(* IEC 61131-3 sources: volt/packages/volt-lsp-iec/test-corpus/bakon-nano/Device/Plc Logic/Application/Global Variables, 9 files *)

(* ---- CAN_TO_PLC.gvl ---- *)
//This gobal variable list is received via the network.
//Sender: Imported from file '\\SRV2012\Home$\pieter\Documents\Projecten\P10037 Hert nano met wasbak\21000149 Software\CAN Bridge\CAN_TO_PLC.gvl'
//Protocol: UDP

{attribute 'qualified_only'}
VAR_GLOBAL
	dwAGM1_PowerLoss			: DWORD;
	rAGM1_Frequency				: REAL;
	bAGM1_CommFailure			: BOOL;
	dwErrorDetailsAGM1			: DWORD;
	bUltrasonic1				: BOOL;
END_VAR
%CLASS NVL
%NETVAR ImportFromFile: true
%NETVAR ImportFileName: \\SRV2012\Home$\pieter\Documents\Projecten\P10037 Hert nano met wasbak\21000149 Software\CAN Bridge\CAN_TO_PLC.gvl
%NETVAR TaskName: LogicTask
%NETVAR SenderGVLName: ''
%NETVAR ImportNetVarProperties.Acknowledge: false
%NETVAR ImportNetVarProperties.Checksum: false
%NETVAR ImportNetVarProperties.EventVariable: ''
%NETVAR ImportNetVarProperties.Interval: T#50ms
%NETVAR ImportNetVarProperties.ListIdentifier: 2
%NETVAR ImportNetVarProperties.MinimumGap: T#20ms
%NETVAR ImportNetVarProperties.PackVariables: true
%NETVAR ImportNetVarProperties.ProtocolName: UDP
%NETVAR ImportNetVarProperties.TransmitCyclic: true
%NETVAR ImportNetVarProperties.TransmitOnChange: false
%NETVAR ImportNetVarProperties.TransmitOnEvent: false
%NETVAR ImportNetVarProperties.TaskName: LogicTask
%NETVAR ImportNetVarProperties.ImportFileName: ''
%NETVAR ImportNetVarProperties.ProtocolParameterValues: UDP=Broadcast Adr.=192.168.27.230; Port=1202

(* ---- Global_Constantes_MachineDependant.gvl ---- *)
VAR_GLOBAL CONSTANT

(*********************** AFHANKELIJK VAN MACHINE!! ***********************)

	C_LimitKnifeStrokeMax		: REAL := 225;		(* Controle of machine parameter tussen de limieten valt *)
	C_LimitKnifeStrokeMin		: REAL := 60;		(* (controle of mach par goed opgeslagen zijn) *)

	C_rTargetX_TableCheck		: REAL := 2.1;		(* x positie voor de tafel sensor controle *)
	C_rXAxis_SafeCleaningPos	: REAL := 3;		(* x positie voor de tafel veilig om waterbakje omhoog te sturen *)

	C_rExtraMarginKnifeHeight	: REAL := 8;		(* extra starthoogte van het mes bovenop de gewenste producthoogte *)

	C_rMinOvershootX			: REAL	:= 3;		(* minimaal 1 meer dan de negatieve sw limit *)
	C_rMaxOvershootX			: REAL	:= 683;//688	(* minimaal 1 minder dan de positieve sw limit *)
	C_rMaxOvershootX_XL			: REAL  := 898;		(* voor XL Machine*)
	C_rMinOvershootY			: REAL	:= 3;		(* minimaal 1 meer dan de negatieve sw limit *)
	C_rMaxOvershootY			: REAL	:= 488;		(* minimaal 1 minder dan de positieve sw limit *)
	C_rMaxOvershootY_XL			: REAL  := 658;

	C_rMinimumTrimSlab		: REAL	:= 0;
	C_rMaxPowerUS1			: REAL	:= 100;		(* value from 50 to 100 % *)

	(********************************************* Other  Constantes *********************************************)
	C_rPi								: REAL	:= 3.14159265358979;

	C_wNumberOfMotionObjects	: INT := 1600;

	C_NOT_ACTIVE  				:INT	:=  -1;
	C_INITIAL      					:INT	:=   0;
	C_WAIT_EXEC  	  			:INT	:=	995;
	C_INITIALISE   				:INT 	:=	996;
	C_STOPPED      				:INT	:=	997;
	C_READY        				:INT	:=	998;
	C_LAST       	  				:INT	:=	999;

END_VAR

(* ---- Global_Variables.gvl ---- *)
	VAR_GLOBAL
	g_sMACH							: sMACH_DATA;

	g_bCMD_US_Start1				: BOOL;
	g_bCMD_US_Test1					: BOOL;
	g_bUS_EnableRV					: BOOL;		(* Enable US generator when knife is in product *)
	g_bUS_EnableCleaning			: BOOL;		(* Enable US generator during cleaning *)

	g_bSaveMachPar					: BOOL;		(* Save Mach par aan einde van automaat *)

	ModusRV							: sModusRondVierkant;

	g_uParRondVierkant				: strRondVierkantParameters;

	g_bFirstCycle					: BOOL;
	g_bOnDelayed					: BOOL;

	g_bCalculationStart				: BOOL;
	g_bCalculationDone				: BOOL;
	g_bSUB_CleanKnifeStart			: BOOL;
	g_bSUB_CleanKnifeDone			: BOOL;
	g_bCleanRequest					: BOOL;

	g_bSUB_InitStart				: BOOL;
	g_bSUB_InitDone					: BOOL;

	g_bProductNotFinished			: BOOL;	(* cuts on product not completed *)

	g_bHomingDone					: BOOL;

	g_bTestAGM1						: BOOL;
	g_bResetMaster					: BOOL;
	(* Machine configuration bits *)
	gMachConfig						: sMach_Setup;
	gProductOption					: sProd_Setup;

	(* Ultrasonic variables *)
	//g_dwAGM1_Status					: DWORD;
	g_dwAGM1_PowerLoss				: DWORD;
	g_rAGM1_Frequency				: REAL;

	g_sCalculated					: sMACH_Calculated;
	g_aCuttingPositions				: ARRAY [1..C_wNumberOfMotionObjects] OF XYA_Target;
	g_sCuttingPositionsInfo			: ArrayInfo;
	g_aWastePositions				: ARRAY [1..100] OF XYA_Target;
	g_sWastePositionsInfo			: ArrayInfo;

	g_bTrimFront					: BOOL;	(* Variable used in calculation functions*)
	g_bTrimRear						: BOOL;	(* Variable used in calculation functions*)
	g_bTrimLeft						: BOOL;	(* Variable used in calculation functions*)
	g_bTrimRight					: BOOL;	(* Variable used in calculation functions*)
	g_rDistanceBetweenCuts_InX		: REAL;	(* Variable used in calculation functions*)
	g_rDistanceBetweenCuts_InY		: REAL;	(* Variable used in calculation functions*)
	g_rHoekInRad					: REAL;	(* Variable used in calculation functions*)
	g_rHoekInRad2					: REAL;	(* Variable used in calculation functions*)
	g_rEndTargetX					: REAL;	(* Variable used for saving end target*)
	g_rEndTargetY					: REAL;	(* Variable used for saving end target*)
	g_rEndTargetA					: REAL;	(* Variable used for saving end target*)
	g_rEndTargetK					: REAL;	(* Variable used for saving end target*)

	g_bCurrentTableUniversal10		: BOOL := FALSE;

	g_sMCHCopyMade					: BOOL := FALSE;
	g_sMCHParCopy					: sMACH_MACH_Parameters;
	g_sRCPCopyMade					: BOOL := FALSE;
	g_sRCPParCopy					: sMACH_RCP_Parameters;
	{warning 'Disabled for compatibility - SVE'}
	//g_Logger						: PLC_Logger;
END_VAR

(* ---- PLC_TO_CAN.gvl ---- *)
{attribute 'qualified_only'}
VAR_GLOBAL
	g_bOnDelayed 			: BOOL;
	g_bDQ_Ultrasonic1 		: BOOL;
	g_bTestAGM1 			: BOOL;
	g_HMI_MCH_Parameters	: sMACH_MACH_Parameters;
	g_HMI_RCP_Parameters	: sMACH_RCP_Parameters;
	g_HMI_MachCommand		: sMACH_HMI_UnitCmd;
	C_rMaxPowerUS1			: REAL;
END_VAR
%NETVAR Acknowledge: false
%NETVAR Checksum: false
%NETVAR EventVariable: ''
%NETVAR Interval: T#50ms
%NETVAR ListIdentifier: 1
%NETVAR MinimumGap: T#20ms
%NETVAR PackVariables: true
%NETVAR ProtocolName: UDP
%NETVAR TransmitCyclic: true
%NETVAR TransmitOnChange: false
%NETVAR TransmitOnEvent: false
%NETVAR TaskName: LogicTask
%NETVAR ImportFileName: ''
%NETVAR ProtocolParameterValues: UDP=Broadcast Adr.=192.168.27.231; Port=1202
%FILE_LINK ExportBeforeCompile '\\SRV2012\Home$$\pieter\Documents\Projecten\P10037 Hert nano met wasbak\21000149 Software\PLC\PLC_TO_CAN.gvl'

(* ---- VAR_AxisControl_ECSEP.gvl ---- *)
VAR_GLOBAL
	g_uControl_X_Axis		:KC_AxisBasicsControl;	(* VIRTUAL AXIS *)
	g_uStatus_X_Axis			:KC_AxisBasicsStatus;	(* VIRTUAL AXIS *)
	g_uControl_Y_Axis		:KC_AxisBasicsControl;	(* VIRTUAL AXIS *)
	g_uStatus_Y_Axis			:KC_AxisBasicsStatus;	(* VIRTUAL AXIS *)
	g_uControl_Front_Axis	:KC_AxisBasicsControl;
	g_uStatus_Front_Axis	:KC_AxisBasicsStatus;
	g_uControl_Rear_Axis	:KC_AxisBasicsControl;
	g_uStatus_Rear_Axis		:KC_AxisBasicsStatus;
	g_uControl_Z_Axis		:KC_AxisBasicsControl;
	g_uStatus_Z_Axis			:KC_AxisBasicsStatus;
	g_uControl_R_Axis		:KC_AxisBasicsControl;
	g_uStatus_R_Axis		:KC_AxisBasicsStatus;
END_VAR

(* ---- VAR_HMI.gvl ---- *)
VAR_GLOBAL
	(* Communicatie met VisiwinNet Visualisatie Professional V6.3 *)
	g_HMI_MachCommand					: sMACH_HMI_UnitCmd;

	g_HMI_bRecipeIsReset		: BOOL;

	(*status variables *)
	g_sHMI_Mach_UnitStatus				:sMACH_HMI_UnitStatus;				(*module status variables*)

	(* Counters *)
	g_sHMI_CountersDay					: sCounters;		(* all day counters *)

	g_sHMI_ScanData					: sScanData;	(*Data for max follow/torque scan of machine*)

	(* Data for new visu *)
	g_sHMI_VisuCutsArray	: ARRAY[1..150] OF VisuCut;
	g_sHMI_NewRecipeName			: STRING;
	g_bHMI_UseExistingRecipe		:BOOL;
	g_sHMI_FromCecipeName			: STRING;
	g_sHMI_MachParName				: STRING;
	g_sHMI_RcpClmns					: ClmnChoices;
	g_sHMI_Recipe_Clmn1_Choice	: INT; // SlabRound = 1, SlabRound with fingers = 2, Tray = 3
	g_sHMI_Recipe_Clmn2_Choice	: INT; //
	g_sHMI_Recipe_Clmn3_Choice	: INT;
	g_sHMI_Recipe_Clmn1_SlabRound_Choices: INT;
	g_sHMI_Recipe_Clmn1_SlabRoundF_Choices: INT;
	g_sHMI_Recipe_Clmn1_Tray_Choices: INT;
	g_sHMI_Recipe_Clmn2_Slab_Choices: INT;
	g_sHMI_Recipe_Clmn2_Round_Choices: INT;
	g_sHMI_Recipe_Clmn2_SlabF_Choices: INT;
	g_sHMI_Recipe_Clmn2_RoundF_Choices: INT;
	g_sHMI_DashboardNotifications : DashboardNotifications;
	g_HMI_RCP_Parameters_Visu					: sMACH_RCP_Parameters;
	g_HMI_RCP_ShowRCPwastesettings		: BOOL;
	g_HMI_RCP_ShowCleaningsettings		: BOOL;
	g_HMI_RCP_ShowCrashDetectionSettings		: BOOL;
	g_HMI_RCP_ActPartSize	: STRING;
	g_HMI_RCP_UseWasteFront : BOOL;
	g_HMI_RCP_UseWasteRear : BOOL;
	g_HMI_RCP_UseWasteLeft : BOOL;
	g_HMI_RCP_UseWasteRight : BOOL;
	g_HMI_OnDashboard		: BOOL;
	g_HMI_bShowOverlay			: BOOL;
	g_HMI_bCloseOverlay			: BOOL;
	g_HMI_bNewRecipe			: BOOL;
END_VAR

(* ---- VAR_HMI_PERSIST.gvl ---- *)
VAR_GLOBAL PERSISTENT RETAIN
	(* recipe variables *)
	g_HMI_sRecipeName 						:STRING :=  'new recipe';

	g_HMI_RCP_Parameters					: sMACH_RCP_Parameters;

(******************************************************************************************************************)
(*machine parameters*)
	g_HMI_MCH_dnBlockCounter			: DINT := 0;

	g_HMI_nDefaultLanguage				: INT := 1031;
	g_HMI_nSecondLanguage				: INT := 1043;

	g_HMI_MCH_Parameters				: sMACH_MACH_Parameters;

	g_HMI_dnLastMaintenance				: DINT;

(* Counters *)
	g_sHMI_CountersInfinite					: sCounters;		(* all infinite counters *)

(* Machine settings *)
	g_HMI_dwMachineConfig		: DWORD := 16#0000;	(* 0000.0000 *)
	(*	Bit 0 = PneumaticAxis in machine 		//Not used anymore
		Bit 1 = Cleaning installation
		Bit 2 = Nano machine, mutually exlusive with XL		//Not used anymore
		Bit 3 = XL machine, mutually exlusive with Nano
		Bit 4 = RedCase enabled *)

	g_HMI_dwProductOptions		: DWORD := 16#0000;	(* 0000.0000 *)
	(*
		Prod_SlabSquare				:= 0,		(* ProductType = 0 = Slab Square *)
		Prod_SlabTriangle			:= 1,		(* ProductType = 1 = Slab triangle *)
		Prod_SlabDiagonal			:= 2,		(* ProductType = 2 = Slab diagonal *)
		Prod_Round					:= 3,		(* ProductType = 3 = Round Cake *)
		Prod_TraySquareSmall		:= 4,		(* ProductType = 4 = Tray Square Small *)
		Prod_TraySquareLarge		:= 5,		(* ProductType = 5 = Tray Square Large *)
		Prod_TraySquareTriple		:= 6,		(* ProductType = 6 = Tray Square 4 on a table *)
		Prod_SlabSquareClamp		:= 7,		(* ProductType = 7 = Slab Square op tafel met opklemvingers (V04.01) *)
		Prod_TraySquareDouble		:= 8,		(* ProductType = 8 = Tray square 2 side by side*)
		Prod_RoundQuatro			:= 9,		(* ProductType = 9 = Round cake 4 off*)
		Prod_SlabDouble				:= 10		(* productType = 10 = Slab double, alleen door te snijden in 90 graden*)

		Triangles In Tray			:= 15		(* Part of producttype 4 and 5 *)
	*)

(* Memory bits for Set ref axis *)
	g_bAxis_RSet			: BOOL;
	g_bAxis_FrontSet		: BOOL;
	g_bAxis_RearSet		: BOOL;

	(*Bits for redcase retry*)
	g_bContactRedCase : BOOL;
	g_bScanDataPending	: BOOL;
	g_bRedCaseTried		: BOOL;
	g_nRedCaseLastTime: DATE_AND_TIME;

	(* Bits for new visualisation *)
	//Operation menu
	g_bShowCurrRecipeName			: BOOL;
	g_bShowNumberOfProdTotal		: BOOL;
	g_bShowNumberOfProdDay			: BOOL;
	g_bShowNumberOfProdHour			: BOOL;
	g_bShowMachineState				: BOOL;

	//Quick Menu
	g_bShowCleaningMode				: BOOL;
	g_bShowRecipes					: BOOL;
	g_bShowManual					: BOOL;
	g_bShowSettings					: BOOL;
	g_bShowAlarms					: BOOL;
	g_bShowCleanKnifeBtn			: BOOL;
	g_bShowProdCount				: BOOL;

END_VAR
%CLASS PERSISTENT

(* ---- VAR_IO_Station.gvl ---- *)
VAR_GLOBAL

	g_byInputs_Module_00						: BYTE;
	g_byInputs_Module_01						: BYTE;
	g_byInputs_Module_02						: BYTE;//Spare
	g_byInputs_Module_03						: BYTE;//Spare
	g_byInputs_Module_04						: BYTE;//Spare
	g_byInputs_Module_05						: BYTE;//Spare
	g_byOutputs_Module_00						: BYTE;
	g_byOutputs_Module_01						: BYTE;
	g_wInputs_Module_00							: WORD;
	g_wInputs_Module_01							: WORD;
	g_wOutputs_Module_00						: WORD;
	g_wOutputs_Module_01						: WORD;

(*digital inputs from CAN remote IO *)
(*first module *)
	g_bDI_ES_DirectOK							: BOOL;
	g_bDI_CircuitBreaker_i700					: BOOL;		(*Laag wanneer de automaat voor de voedingsunit getript is *)
	g_bDI_CircuitBreaker_Ultrasonic				: BOOL;		(*Laag wanneer de automaat voor de ultrasoongenerator eruit ligt*)
	g_bDI_PressureSwitchOK						: BOOL;
	g_bDI_StartButton							: BOOL;
	g_bDI_LightCurtainOK						: BOOL;
	g_bDI_MachineInSafePosition					: BOOL;		(* Feedback from Pilz, table in infeed position and knife up *)
	g_bDI_TableCheck							: BOOL;		(* Sensor for checking if the table correspondents with the recipe *)

(*second module *)
	g_bDI_Servo_Power_OK						: BOOL;
	g_bDI_CleaningContainerUp					: BOOL;		//Spare
	g_bDI_CleaningContainerDown					: BOOL;		//Spare
	g_bDI_UltraSonic_Error						: BOOL;
	g_bDI_UltraSonic_ErrorCode_1				: BOOL;
	g_bDI_UltraSonic_ErrorCode_2				: BOOL;
	g_bDI_Spare16								: BOOL;
	g_bDI_Spare17								: BOOL;

(* Digital outputs *)
(* Third module *)
	g_bDQ_ResetSafety							: BOOL;
	g_bDQ_LightCurtainActive					: BOOL;
	g_bDQ_MainValve								: BOOL;		(* activate airvalve *)
	g_bDQ_Ultrasonic1							: BOOL;
	g_bDQ_LampStart								: BOOL;
	g_bDQ_Servo_Power_Reset						: BOOL;
	g_bDQ_Buzzer								: BOOL;
	g_bDQ_Spare_17								: BOOL;

(* Fourth module *)
	g_bDQ_CleaningContainerUp					: BOOL;
	g_bDQ_CleaningContainerDown					: BOOL;
	g_bDQ_CleaningAirValve						: BOOL;
	g_bDQ_CleaningWaterValve					: BOOL;
	g_bDQ_Spare_24								: BOOL;
	g_bDQ_Spare_25								: BOOL;
	g_bDQ_Spare_26								: BOOL;
	g_bDQ_Spare_27								: BOOL;

(* Analog inputs *)
(* Fifth module *)
	g_iAI_UltrasonicPower						: INT;
	g_iAI_Spare_01								: INT;

(* Analog outputs *)
(* Sixth module *)
	g_iAQ_UltrasonicPower						: INT;
	g_iAQ_Spare_01								: INT;

END_VAR

(* ---- Variable_Configuration.gvl ---- *)
VAR_CONFIG
END_VAR
